TYPE ST_SearchData :
STRUCT
	dtStartTimestamp : DT;
	dtEndTimestamp : DT;
END_STRUCT
END_TYPE

(* stored: Version 1.1.0.1, ProductVersion 3.1.4024.14
   DUT ST_SearchData: Id {a8c614c2-65d4-449b-9a8d-e8e8c9df32fb} *)
